Universal Robots PolyScope program: tool_contact_test.urp

Program tool_contact_test (installation=default directory=/ursim/programs createdIn=5.21.3 lastSavedIn=5.21.3 robotSerialNumber=20195599999)
Calibrated DH parameters: a=[0, -0.425, -0.3922, 0, 0, 0]; d=[0.1625, 0, 0, 0.1333, 0.0997, 0.0996]; alpha=[1.570796, 0, 0, 1.570796, -1.570796, 0]; deltaTheta=[0, 0, 0, 0, 0, 0]
InitVariablesNode
Robot Program (runOnlyOnce=false)
  MoveL speed 250 mm/s, acceleration 1200 mm/s^2 (useActiveTCP=true optimoveEnabled=false optiMoveSpeed=0.3 optiMoveAcceleration=0.09) feature=Base
    Waypoint Waypoint_1: TCP in base x=55.247 y=-644.966 z=101.33 mm, rx=1.5508 ry=0.228 rz=0.2298 rad; joints [-73.211, -129.398, -98.431, -131.721, 270.063, -0.002] deg
    MoveDirectionNode (selectedDirection=XPlus toolParams=0.03, 1.2) feature=Joint_6_name
      Until TOOL_CONTACT_DETECTION (allowActions=true retraction=0.005 decelerationAcceleration=3 decelerationAngularAcceleration=34.906585)
        var_1 := get_actual_tcp_pose()
  MoveL speed 250 mm/s, acceleration 1200 mm/s^2 (useActiveTCP=true optimoveEnabled=false optiMoveSpeed=0.3 optiMoveAcceleration=0.09) feature=Base
    Waypoint Waypoint_2: TCP in base x=55.247 y=-745.808 z=101.33 mm, rx=1.5508 ry=0.228 rz=0.2298 rad; joints [-75.843, -139.686, -77.532, -142.332, 267.43, 0.019] deg
    MoveDirectionNode (selectedDirection=XPlus toolParams=0.03, 1.2) feature=Joint_6_name
      Until TOOL_CONTACT_DETECTION (allowActions=true retraction=0.005 decelerationAcceleration=3 decelerationAngularAcceleration=34.906585)
        var_2 := get_actual_tcp_pose()
